FUNCTION_BLOCK FC_Observer (* State observer: one coherent Cell snapshot; invalid or unsafe states inhibit skills *)
  (* Standard: 61499-2 *)
  (* Version 2.0, 2026-09-27, Project contributors, Filling cell reference model *)
  PACKAGE fillingcell;
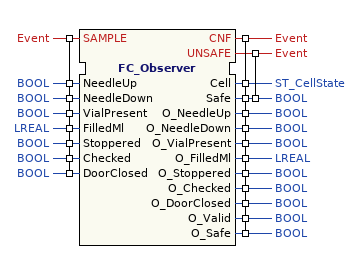
  EVENT_INPUT
    SAMPLE WITH NeedleUp, NeedleDown, VialPresent, FilledMl, Stoppered, Checked, DoorClosed;
  END_EVENT
  EVENT_OUTPUT
    CNF WITH Cell, Safe, O_NeedleUp, O_NeedleDown, O_VialPresent, O_FilledMl, O_Stoppered, O_Checked, O_DoorClosed, O_Valid, O_Safe;
    UNSAFE WITH Safe;
  END_EVENT
  VAR_INPUT
    NeedleUp : BOOL;
    NeedleDown : BOOL;
    VialPresent : BOOL;
    FilledMl : LREAL;
    Stoppered : BOOL;
    Checked : BOOL;
    DoorClosed : BOOL;
  END_VAR
  VAR_OUTPUT
    Cell : fillingcell::ST_CellState;
    Safe : BOOL;
    O_NeedleUp : BOOL;
    O_NeedleDown : BOOL;
    O_VialPresent : BOOL;
    O_FilledMl : LREAL;
    O_Stoppered : BOOL;
    O_Checked : BOOL;
    O_DoorClosed : BOOL;
    O_Valid : BOOL;
    O_Safe : BOOL;
  END_VAR
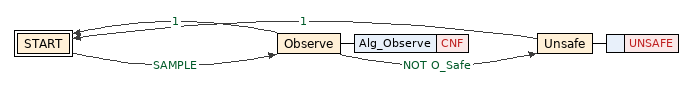
  EC_STATES
    START;
    Observe : Alg_Observe -> CNF;
    Unsafe : -> UNSAFE;
  END_STATES
  EC_TRANSITIONS
    START TO Observe := SAMPLE;
    Observe TO Unsafe := NOT O_Safe;
    Observe TO START := 1;
    Unsafe TO START := 1;
  END_TRANSITIONS
  ALGORITHM Alg_Observe IN ST:
O_NeedleUp := NeedleUp;
O_NeedleDown := NeedleDown;
O_VialPresent := VialPresent;
O_FilledMl := FilledMl;
O_Stoppered := Stoppered;
O_Checked := Checked;
O_DoorClosed := DoorClosed;
O_Valid := (FilledMl >= 0.0) AND NOT (NeedleUp AND NeedleDown);
O_Safe := O_Valid AND DoorClosed;
Cell.NeedleUp := O_NeedleUp;
Cell.NeedleDown := O_NeedleDown;
Cell.VialPresent := O_VialPresent;
Cell.FilledMl := O_FilledMl;
Cell.Stoppered := O_Stoppered;
Cell.Checked := O_Checked;
Cell.DoorClosed := O_DoorClosed;
Cell.Valid := O_Valid;
Cell.Safe := O_Safe;
Safe := O_Safe;
  END_ALGORITHM
END_FUNCTION_BLOCK
